FUNCTION_BLOCK FB_OPCUA_WorkOnNode IMPLEMENTS I_OPCUA_WorkOnNode
VAR_INPUT
END_VAR
VAR_OUTPUT
	busy: BOOL;
	error : BOOL;
END_VAR
VAR

	stNodeAddInfo			: ST_UANodeAdditionalInfo;
	cbData_R				: UDINT;
	
	iState		: INT;
	nErrorID	: DWORD;
	dataAdd : PVOID;
	lastErrorStep: INT;
	Executing : BOOL;
	writeStep : INT;
	(* Declarations for UA_Write *)
	{IF defined (Test)}
		_iOPCUA_Write : I_OPCUA_Write; 
		(* Declarations for UA_NodeReleaseHandle *)
		_iOPCUA_NodeReleaseHandle : I_OPCUA_NodeReleaseHandle;
		_iOPCUA_NodeGetHandle : I_OPCUA_NodeGetHandle;
		_iOPCUA_Read			: I_OPCUA_Read;
	{ELSE}
		_iOPCUA_Write : UA_WriteWrapper;
		_iOPCUA_NodeReleaseHandle : UA_NOdeReleaseHandleWrapper;
		_iOPCUA_NodeGetHandle : UA_NodeGetHandleWrapper;
		_iOPCUA_Read			: UA_ReadWrapper;
	{ END_IF}
	(* Other declarations *) 
	errorID : DWORD;	
	clientVariablePrev : BYTE;
	firstTimeWrite : BOOL;
	//_iOPCUA_NodeGetHandle : I_OPCUA_NodeGetHandle;
	NodeID : ST_UANodeID;
	nNodeHdl : DWORD;
	NodeGetHandleBusy: BOOL;
	NodeGetHandleError: BOOL;
	NodeGetHandleErrorID: DWORD;
	readBusy: BOOL;
	readError: BOOL;
	readErrorID: DWORD;
	nodeReleaseHandleBusy: BOOL;
	nodeReleaseHandleError: BOOL;
	nodeReleaseHandleErrorID: DWORD;
	writeBusy: BOOL;
	writeError: BOOL;
	writeErrorID: DWORD;
	clientVarInfo : __SYSTEM.VAR_INFO;
	pClientByteValue : POINTER TO BYTE;
	ConnectionHdlPrev: DWORD;
END_VAR

METHOD FB_init : BOOL
VAR_INPUT
	bInitRetains : BOOL; // if TRUE, the retain variables are initialized (warm start / cold start)
	bInCopyCode : BOOL;  // if TRUE, the instance afterwards gets moved into the copy code (online change)
	{IF defined (Test)}
		iOPCUA_Write				: I_OPCUA_Write;
		iOPCUA_Read					: I_OPCUA_Read;
		iOPCUA_NodeReleaseHandle 	: I_OPCUA_NodeReleaseHandle;
		iOPCUA_NodeGetHandle 		: I_OPCUA_NodeGetHandle;
	{END_IF}
END_VAR
{IF defined (Test)}
	_iOPCUA_Write	:= iOPCUA_Write;		
	_iOPCUA_Read		:= iOPCUA_Read	;		
	_iOPCUA_NodeReleaseHandle := iOPCUA_NodeReleaseHandle;
	_iOPCUA_NodeGetHandle 	:= iOPCUA_NodeGetHandle 	;
{END_IF}
END_METHOD

{warning 'add method implementation '}
METHOD read : BOOL
VAR_INPUT
	{attribute 'anytypeclass' := 'ANY'}
	//clientVariable	: ANY;
	(* VAR_INFO of the target variable (from GVL_OPC)*)
	//clientVariableInfo	: __SYSTEM.VAR_INFO;
	clientVariableAddress : PVOID;
	clientVariableSize : UDINT;
	serverNodeIdentifier	: STRING;
	nameSpaceLocationIdentifierEx	: STRING(MAX_STRING_LENGTH);
	ConnectionHdl	: DWORD;
	nNamespaceIndex			: UINT;
END_VAR

IF ConnectionHdl <> ConnectionHdlPrev THEN
	istate := 0;
	ConnectionHdlPrev := ConnectionHdl;
	error := FALSE;
END_IF

CASE istate OF
0: 
		error := FALSE;
		nNodeHdl :=0;
		iState := iState + 1;
		Executing := TRUE;
	
1:	(* Get Node Handle *)
	
		NodeID.eIdentifierType := eUAIdentifierType_String;
		NodeID.nNamespaceIndex := nNamespaceIndex;
		NodeID.sIdentifier := CONCAT(nameSpaceLocationIdentifierEx,serverNodeIdentifier);
		_iOPCUA_NodeGetHandle.start(
									Execute := TRUE,
									ConnectionHdl := connectionHdl,
									NodeID := NodeID,
									Timeout := T#5S,
									NodeHdl => nNodeHdl,
									Busy => NodeGetHandleBusy,
									Error => NodeGetHandleError,
									ErrorID => NodeGetHandleErrorID
									);
		IF NOT NodeGetHandleBusy THEN
		  _iOPCUA_NodeGetHandle.start(Execute := FALSE,
										ConnectionHdl := connectionHdl,
										NodeID := NodeID,
										Timeout := T#5S
										);
		  IF NOT NodeGetHandleError THEN
			istate := istate + 1;
		  ELSE
			errorID := NodeGetHandleErrorID;
			istate := 3;
		  END_IF
		END_IF

	
2: 	(* UA_Read *)

	//dataAdd := ADR(clientVariable);
	clientVarInfo := __VARINFO(clientVariableAddress);
	_iOPCUA_Read.start(
						Execute := TRUE,
						ConnectionHdl := connectionHdl,
						NodeHdl := nNodeHdl,
						cbData := clientVariableSize,//clientVarInfo.BitSize,//SIZEOF(clientVariable),//clientVariableInfo.BitSize,
						stNodeAddInfo 	:= stNodeAddInfo,
						pVariable := clientVariableAddress,//clientVariableInfo.ByteAddress,
						Timeout := T#5S,
						busy => readBusy,
						error => readError,
						errorID => readErrorID,
						cbData_R => cbData_R
						);

	IF NOT readBusy THEN
			_iOPCUA_Read.start( Execute := FALSE, 
						ConnectionHdl := connectionHdl,
						NodeHdl := nNodeHdl,
						cbData := clientVarInfo.BitSize,//SIZEOF(clientVariable),//clientVariableInfo.BitSize,
						stNodeAddInfo 	:= stNodeAddInfo,
						pVariable :=clientVariableAddress,//clientVariableInfo.ByteAddress,
						Timeout := T#5S,
						cbData_R => cbData_R);

		IF NOT readError THEN
			iState 		:= 3;
		ELSE
			lastErrorStep := 2;
			nErrorID	:= readErrorId;
			iState 		:= 3; (* idle *)
		END_IF
	END_IF


3:	(* Release Node Handle *)
		_iOPCUA_NodeReleaseHandle.start(
			Execute			:= TRUE,
			ConnectionHdl	:= ConnectionHdl,
			NodeHdl			:= nNodeHdl,
			Timeout := T#5S,
			busy => nodeReleaseHandleBusy,
			error => nodeReleaseHandleError,
			errorID => nodeReleaseHandleErrorID
		);
	
		IF NOT nodeReleaseHandleBusy THEN
			_iOPCUA_NodeReleaseHandle.start(Execute := FALSE,
											ConnectionHdl	:= ConnectionHdl,
											NodeHdl			:= nNodeHdl,
											Timeout := T#5S
											);
	
			IF NOT nodeReleaseHandleError THEN
				Executing := FALSE;
				istate := 0;
			ELSE
				error := TRUE;
				errorID	:= nodeReleaseHandleErrorID;
				istate 	:= 0; (* idle *)
			END_IF
		END_IF
END_CASE
busy := Executing;
END_METHOD

{warning 'add method implementation '}
METHOD write : BOOL
VAR_INPUT
	{attribute 'anytypeclass' := 'ANY'}
	//clientVariable	: ANY;
	(* VAR_INFO of the target variable (from GVL_OPC)*)
	//clientVariableInfo	: __SYSTEM.VAR_INFO;
	clientVariableAddress	: PVOID;
	clientVariableSize : UDINT;
	serverNodeIdentifier	: STRING;
	nameSpaceLocationIdentifierEx	: STRING(MAX_STRING_LENGTH);
	connectionHdl: DWORD;
	nNamespaceIndex			: UINT;
END_VAR

IF ConnectionHdl <> ConnectionHdlPrev THEN
	writeStep := 0;
	ConnectionHdlPrev := ConnectionHdl;
	error := FALSE;
	firstTimeWrite := FALSE;
END_IF

CASE writeStep OF
	
	0:
		error := FALSE;
		clientVarInfo := __VARINFO(clientVariableAddress);
		pClientByteValue := clientVariableAddress;
		nNodeHdl := 0;
		//MEMSET(ADR(clientByteValue), clientVarInfo.ByteAddress ,clientVarInfo.BitSize);
		//IF clientVariable.pValue^ <> clientVariablePrev OR NOT firstTimeWrite THEN
		IF pClientByteValue^ <> clientVariablePrev OR NOT firstTimeWrite THEN
			Executing := TRUE;
			clientVariablePrev := pClientByteValue^;
			writeStep := 1;
		END_IF
	
	  1: 
		(* UA_NodeGetHandle *)
		NodeID.eIdentifierType := eUAIdentifierType_String;
		NodeID.nNamespaceIndex := nNamespaceIndex;
		NodeID.sIdentifier := CONCAT(nameSpaceLocationIdentifierEx,serverNodeIdentifier);
		_iOPCUA_NodeGetHandle.start(
									Execute := TRUE,
									ConnectionHdl := connectionHdl,
									NodeID := NodeID,
									Timeout := T#5S,
									NodeHdl => nNodeHdl,
									Busy => nodeGetHandleBusy,
									Error => nodeGetHandleError,
									ErrorID => nodeGetHandleErrorID
									
									);
		IF NOT nodeGetHandleBusy THEN
		  _iOPCUA_NodeGetHandle.start(Execute := FALSE,
									ConnectionHdl := connectionHdl,
									NodeID := NodeID,
									Timeout := T#5S,);
		  IF NOT nodeGetHandleError THEN
			writeStep := writeStep + 1;
		  ELSE
			errorID := nodeGetHandleErrorID;
			writeStep := 2;
		  END_IF
		END_IF
	  2: (* UA_Write *)
		_iOPCUA_Write.start(
							Execute := TRUE,
							ConnectionHdl := connectionHdl,
							NodeHdl := nNodeHdl,
							stNodeAddInfo := stNodeAddInfo,
							cbData := clientVariableSize,//clientVarInfo.BitSize,//SIZEOF(clientVariable),//clientVariableInfo.BitSize,
							pVariable := clientVariableAddress,//clientVariableInfo.ByteAddress,
							Timeout := T#5S,
							busy => writeBusy,
							error => writeError,
							errorID => writeErrorID
							);
		IF NOT writeBusy THEN
		  _iOPCUA_Write.start(
								Execute := FALSE,
								ConnectionHdl := connectionHdl,
								NodeHdl := nNodeHdl,
								stNodeAddInfo := stNodeAddInfo,
								cbData := clientVarInfo.BitSize,//SIZEOF(clientVariable), //clientVariableInfo.BitSize,
								pVariable := clientVariableAddress,//clientVariableInfo.ByteAddress,
								Timeout := T#5S );

		  IF NOT writeError THEN
				writeStep := 3;
		  ELSE
			//Executing := FALSE;
			//error := TRUE;
			errorID := writeErrorID;
			writeStep := 3;
		  END_IF
		END_IF
	3:	(* Release Node Handle *)
		_iOPCUA_NodeReleaseHandle.start(
			Execute			:= TRUE,
			ConnectionHdl	:= ConnectionHdl,
			NodeHdl			:= nNodeHdl,
			TimeOut			:= T#5S,
			Busy			=> nodeReleaseHandleBusy,
			Error			=> nodeReleaseHandleError,
			ErrorID			=> nodeReleaseHandleErrorID
		);
	
		IF NOT nodeReleaseHandleBusy THEN
			_iOPCUA_NodeReleaseHandle.start(Execute := FALSE,
											ConnectionHdl	:= ConnectionHdl,
											NodeHdl			:= nNodeHdl,
											TimeOut			:= T#5S
												);
	
			IF NOT nodeReleaseHandleError THEN
				firstTimeWrite := TRUE;
				Executing := FALSE;
				writeStep := 0;
			ELSE
				error := TRUE;
				errorID	:= nodeReleaseHandleErrorID;
				writeStep 	:= 0; (* idle *)
			END_IF
		END_IF
END_CASE
busy := Executing ;
END_METHOD

END_FUNCTION_BLOCK

(* stored: Version 1.1.0.1, ProductVersion 3.1.4024.9
   POU FB_OPCUA_WorkOnNode: Id {0e3c7aeb-71ed-4c55-86bf-e2c7680b355d}, SpecialFunc None
   Method FB_init: Id {e3f5c172-5b53-41bb-83ce-9b70c20f0d0c}
   Method read: Id {03c3b3f3-09be-48e8-a71a-d9f38d3c1c07}
   Method write: Id {64b5c044-7dd9-4728-a1be-b684ca04e6b0} *)
